(* IEC 61131-3 sources: SJ_AGV/PLC/Standard_functions.4.4.0/Safety, 2 files *)

(* ---- ASCII_TO_DEC.ST ---- *)
FUNCTION_BLOCK ASCII_TO_DEC
VAR_EXTERNAL

END_VAR

VAR_INPUT
	ASCII : dint;
END_VAR

VAR CONSTANT
	ASCII_a61 	: DINT := 16#61; 	(* Chr "a" *)
	ASCII_A41 	: DINT := 16#41; 	(* Chr "A" *)
	ASCII_0 	: DINT := 16#30;	(* Number "0" *)
END_VAR

VAR_OUTPUT
	dec	: dint;
END_VAR

VAR
	CODE : DINT;
END_VAR
IF 		ASCII >= ASCII_a61 THEN		(* Character a *)
	dec := ASCII - ASCII_a61 + 10;

elsif 	ASCII >= ASCII_A41 THEN	(* Character A *)
	dec := ASCII - ASCII_A41 + 10;

else
	dec := ASCII - ASCII_0;			(* Number *)
END_IF;

END_FUNCTION_BLOCK

(* ---- DRIVERSUPERVISION_FB.ST ---- *)
FUNCTION_BLOCK DRIVERSUPERVISION_FB
VAR_EXTERNAL
	NDC8 : NDC8_T;

END_VAR

VAR_INPUT
	Command : INT;
	FeedBack : INT;
	Range : INT;
	Timeout : TIME;
	Moving : BOOL;

END_VAR

VAR_OUTPUT
	OverRangeFail : BOOL;
	NotMovingFail : BOOL;
END_VAR

VAR
	iFeedBack : INT;
	Diff : INT;

	OverRange_failure : BOOL;
	NotMoving_failure : BOOL;

	MovingR : R_Trig;
	MovingF : F_Trig;

	OverRangeFailTimerTON : TON;
	NotMovingFailTimerTON : TON;

END_VAR
OverRangeFailTimerTON(IN:=OverRange_failure, Pt:=Timeout);
NotMovingFailTimerTON(IN:=NotMoving_failure, Pt:=Timeout);

MovingR(CLK:= Moving);
MovingF(CLK:= Moving);

if MovingF.Q then
	OverRangeFailTimerTON(IN := FALSE);
	NotMovingFailTimerTON(IN := FALSE);

	NotMoving_failure := FALSE;
	OverRange_failure := FALSE;

	OverRangeFail := FALSE;
	NotMovingFail := FALSE;
end_if;

if MovingR.Q then
	iFeedBack := FeedBack;
end_if;

Diff := FeedBack - Command;

if abs(Diff) > Range then
	OverRange_failure := TRUE;
else
	OverRange_failure := FALSE;
end_if;

if OverRangeFailTimerTON.Q = TRUE then
	OverRangeFail := TRUE;
else
	OverRangeFail := FALSE;
end_if;

if Moving then
	if FeedBack = iFeedBack then
		NotMoving_failure:= TRUE;
	else
		NotMoving_failure := FALSE;
	end_if;

	if NotMovingFailTimerTON.Q = TRUE then
		NotMovingFail := TRUE;
	else
		NotMovingFail := FALSE;
	end_if;
end_if;

END_FUNCTION_BLOCK
